// TwinCAT 3 PLC project GattSim
// ProgramVersion: 3.1.4022.3
// libraries:
//   Tc2_Standard, * (Beckhoff Automation GmbH)
//   Tc2_System, * (Beckhoff Automation GmbH)
//   Tc2_Utilities, * (Beckhoff Automation GmbH)
//   Tc3_Module, * (Beckhoff Automation GmbH)
//   Vacuum System Simulator Library, * (SLAC)
// project tree:
//   GVLs/ GVL_GATT.TcGVL, GVL_Variables.TcGVL
//   / PlcTask.TcTTO, SimTask.TcTTO
//   POUs/ MAIN.TcPOU, PRG_DIAGNOSTIC.TcPOU, PRG_GATT.TcPOU
// (motion and I/O tree: see PLC project gattplc)
// real-time tasks:
//   TASK PlcTask: cycle T#10ms, priority 20, ADS port 350
//   TASK SimTask: cycle T#10ms, priority 21, ADS port 351

CONFIGURATION GattSim
    RESOURCE PLC ON TwinCAT3
        TASK PlcTask(INTERVAL := T#10ms, PRIORITY := 20);
        TASK SimTask(INTERVAL := T#10ms, PRIORITY := 21);
        PROGRAM MAIN WITH SimTask : MAIN;
    END_RESOURCE
END_CONFIGURATION

// ---- GVLs/GVL_GATT.TcGVL
VAR_GLOBAL


// ST_Volume

st_AT1K0_GAS_VRC_10_VOL : ST_Volume := (rVolume := 1E3, rPressure := Global_Pressure, rVLeak := Global_Leak);
st_AT1K0_GAS_PTM_10_VOL : ST_Volume := (rVolume := 1E3, rPressure := Global_Pressure, rVLeak := Global_Leak);
st_GATT : ST_Volume := (rVolume := 1E3, rPressure := Global_Pressure, rVLeak := Global_Leak);
st_AT1K0_GAS_VRC_20_VOL : ST_Volume := (rVolume := 1E3, rPressure := Global_Pressure, rVLeak := Global_Leak);
st_AT1K0_GAS_VRC_30_VOL : ST_Volume := (rVolume := 1E3, rPressure := Global_Pressure, rVLeak := Global_Leak);
st_AT1K0_GAS_VRC_40_VOL : ST_Volume := (rVolume := 1E3, rPressure := Global_Pressure, rVLeak := Global_Leak);
st_AT1K0_GAS_VRC_50_VOL : ST_Volume := (rVolume := 1E3, rPressure := Global_Pressure, rVLeak := Global_Leak);
st_AT1K0_GAS_VGP_80_VOL : ST_Volume := (rVolume := 1E3, rPressure := Global_Pressure, rVLeak := Global_Leak);
st_BypassLine2 : ST_Volume := (rVolume := 1E3, rPressure := Global_Pressure, rVLeak := Global_Leak);
st_BypassLine1 : ST_Volume := (rVolume := 1E3, rPressure := Global_Pressure, rVLeak := Global_Leak);
st_AT1K0_GAS_VRC_100_VOL : ST_Volume := (rVolume := 1E3, rPressure := Global_Pressure, rVLeak := Global_Leak);
st_AT1K0_GAS_VRC_110_VOL : ST_Volume := (rVolume := 1E3, rPressure := Global_Pressure, rVLeak := Global_Leak);
st_AT1K0_GAS_PTM_120_VOL : ST_Volume := (rVolume := 1E3, rPressure := Global_Pressure, rVLeak := Global_Leak);
st_AT1K0_GAS_VRC_120_VOL : ST_Volume := (rVolume := 1E3, rPressure := Global_Pressure, rVLeak := Global_Leak);
st_AT1K0_GAS_VRC_130_VOL : ST_Volume := (rVolume := 1E3, rPressure := Global_Pressure, rVLeak := Global_Leak);
st_AT1K0_GAS_PTM_140_VOL : ST_Volume := (rVolume := 1E3, rPressure := Global_Pressure, rVLeak := Global_Leak);
st_AT1K0_GAS_VRC_140_VOL : ST_Volume := (rVolume := 1E3, rPressure := Global_Pressure, rVLeak := Global_Leak);

// ST_MechPump

st_AT1K0_GAS_PTM_10 : ST_MechPump := (iMaxSpd:=1000, rBasePress:=1E-9, rMaxLoad:=0.95);
st_AT1K0_GAS_PTM_20 : ST_MechPump := (iMaxSpd:=1000, rBasePress:=1E-9, rMaxLoad:=0.95);
st_AT1K0_GAS_PMF_10 : ST_MechPump := (rMRE:=10, rBasePress:=1E-3);
st_AT1K0_GAS_PTM_30 : ST_MechPump := (iMaxSpd:=1000, rBasePress:=1E-9, rMaxLoad:=0.95);
st_AT1K0_GAS_PTM_40 : ST_MechPump := (iMaxSpd:=1000, rBasePress:=1E-9, rMaxLoad:=0.95);
st_AT1K0_GAS_PMF_60 : ST_MechPump := (rMRE:=10, rBasePress:=1E-3);
st_AT1K0_GAS_PTM_80 : ST_MechPump := (iMaxSpd:=1000, rBasePress:=1E-9, rMaxLoad:=0.95);
st_AT1K0_GAS_PTM_110 : ST_MechPump := (iMaxSpd:=1000, rBasePress:=1E-9, rMaxLoad:=0.95);
st_AT1K0_GAS_PTM_120 : ST_MechPump := (iMaxSpd:=1000, rBasePress:=1E-9, rMaxLoad:=0.95);
st_AT1K0_GAS_PTM_130 : ST_MechPump := (iMaxSpd:=1000, rBasePress:=1E-9, rMaxLoad:=0.95);
st_AT1K0_GAS_PTM_140 : ST_MechPump := (iMaxSpd:=1000, rBasePress:=1E-9, rMaxLoad:=0.95);

// FB_TurboPump

fb_AT1K0_GAS_PTM_10 : FB_TurboPump;
fb_AT1K0_GAS_PTM_20 : FB_TurboPump;
fb_AT1K0_GAS_PTM_30 : FB_TurboPump;
fb_AT1K0_GAS_PTM_40 : FB_TurboPump;
fb_AT1K0_GAS_PTM_80 : FB_TurboPump;
fb_AT1K0_GAS_PTM_110 : FB_TurboPump;
fb_AT1K0_GAS_PTM_120 : FB_TurboPump;
fb_AT1K0_GAS_PTM_130 : FB_TurboPump;
fb_AT1K0_GAS_PTM_140 : FB_TurboPump;

// ST_VacuumValve

st_AT1K0_GAS_VRC_10 : ST_VacuumValve := (q_xClsLS := TRUE, q_xOpnLS := FALSE);
st_AT1K0_GAS_VRC_20 : ST_VacuumValve := (q_xClsLS := TRUE, q_xOpnLS := FALSE);
st_AT1K0_GAS_VRC_30 : ST_VacuumValve := (q_xClsLS := TRUE, q_xOpnLS := FALSE);
st_AT1K0_GAS_VRC_40 : ST_VacuumValve := (q_xClsLS := TRUE, q_xOpnLS := FALSE);
st_AT1K0_GAS_VRC_50 : ST_VacuumValve := (q_xClsLS := TRUE, q_xOpnLS := FALSE);
st_AT1K0_GAS_VRC_60 : ST_VacuumValve := (q_xClsLS := TRUE, q_xOpnLS := FALSE);
st_AT1K0_GAS_VRC_90 : ST_VacuumValve := (q_xClsLS := TRUE, q_xOpnLS := FALSE);
st_AT1K0_GAS_VRC_100 : ST_VacuumValve := (q_xClsLS := TRUE, q_xOpnLS := FALSE);
st_AT1K0_GAS_VRC_110 : ST_VacuumValve := (q_xClsLS := TRUE, q_xOpnLS := FALSE);
st_AT1K0_GAS_VRC_120 : ST_VacuumValve := (q_xClsLS := TRUE, q_xOpnLS := FALSE);
st_AT1K0_GAS_VRC_130 : ST_VacuumValve := (q_xClsLS := TRUE, q_xOpnLS := FALSE);
st_AT1K0_GAS_VRC_140 : ST_VacuumValve := (q_xClsLS := TRUE, q_xOpnLS := FALSE);

// FB_VacuumValve

fb_AT1K0_GAS_VRC_10 : FB_VacuumValve;
fb_AT1K0_GAS_VRC_20 : FB_VacuumValve;
fb_AT1K0_GAS_VRC_30 : FB_VacuumValve;
fb_AT1K0_GAS_VRC_40 : FB_VacuumValve;
fb_AT1K0_GAS_VRC_50 : FB_VacuumValve;
fb_AT1K0_GAS_VRC_60 : FB_VacuumValve;
fb_AT1K0_GAS_VRC_90 : FB_VacuumValve;
fb_AT1K0_GAS_VRC_100 : FB_VacuumValve;
fb_AT1K0_GAS_VRC_110 : FB_VacuumValve;
fb_AT1K0_GAS_VRC_120 : FB_VacuumValve;
fb_AT1K0_GAS_VRC_130 : FB_VacuumValve;
fb_AT1K0_GAS_VRC_140 : FB_VacuumValve;

// ST_MKS_275

st_AT1K0_GAS_GPI_10 : ST_MKS_275 := (q_xGaugeConnected := TRUE);
st_AT1K0_GAS_GPI_20 : ST_MKS_275 := (q_xGaugeConnected := TRUE);
st_AT1K0_GAS_GPI_11 : ST_MKS_275 := (q_xGaugeConnected := TRUE);
st_AT1K0_GAS_GPI_30 : ST_MKS_275 := (q_xGaugeConnected := TRUE);
st_AT1K0_GAS_GPI_40 : ST_MKS_275 := (q_xGaugeConnected := TRUE);
st_AT1K0_GAS_GPI_50 : ST_MKS_275 := (q_xGaugeConnected := TRUE);
st_AT1K0_GAS_GPI_60 : ST_MKS_275 := (q_xGaugeConnected := TRUE);
st_AT1K0_GAS_GPI_51 : ST_MKS_275 := (q_xGaugeConnected := TRUE);
st_AT1K0_GAS_GPI_80 : ST_MKS_275 := (q_xGaugeConnected := TRUE);
st_AT1K0_GAS_GPI_90 : ST_MKS_275 := (q_xGaugeConnected := TRUE);
st_AT1K0_GAS_GPI_100 : ST_MKS_275 := (q_xGaugeConnected := TRUE);
st_FEES_GATT_GPI_111 : ST_MKS_275 := (q_xGaugeConnected := TRUE);
st_AT1K0_GAS_GPI_110 : ST_MKS_275 := (q_xGaugeConnected := TRUE);
st_AT1K0_GAS_GPI_121 : ST_MKS_275 := (q_xGaugeConnected := TRUE);
st_AT1K0_GAS_GPI_120 : ST_MKS_275 := (q_xGaugeConnected := TRUE);
st_AT1K0_GAS_GPI_130 : ST_MKS_275 := (q_xGaugeConnected := TRUE);
st_AT1K0_GAS_GPI_141 : ST_MKS_275 := (q_xGaugeConnected := TRUE);
st_AT1K0_GAS_GPI_140 : ST_MKS_275 := (q_xGaugeConnected := TRUE);

// FB_MKS_275

fb_AT1K0_GAS_GPI_10 : FB_MKS_275;
fb_AT1K0_GAS_GPI_20 : FB_MKS_275;
fb_AT1K0_GAS_GPI_11 : FB_MKS_275;
fb_AT1K0_GAS_GPI_30 : FB_MKS_275;
fb_AT1K0_GAS_GPI_40 : FB_MKS_275;
fb_AT1K0_GAS_GPI_50 : FB_MKS_275;
fb_AT1K0_GAS_GPI_60 : FB_MKS_275;
fb_AT1K0_GAS_GPI_51 : FB_MKS_275;
fb_AT1K0_GAS_GPI_80 : FB_MKS_275;
fb_AT1K0_GAS_GPI_90 : FB_MKS_275;
fb_AT1K0_GAS_GPI_100 : FB_MKS_275;
fb_FEES_GATT_GPI_111 : FB_MKS_275;
fb_AT1K0_GAS_GPI_110 : FB_MKS_275;
fb_AT1K0_GAS_GPI_121 : FB_MKS_275;
fb_AT1K0_GAS_GPI_120 : FB_MKS_275;
fb_AT1K0_GAS_GPI_130 : FB_MKS_275;
fb_AT1K0_GAS_GPI_141 : FB_MKS_275;
fb_AT1K0_GAS_GPI_140 : FB_MKS_275;

// ST_MKS_422

st_AT1K0_GAS_GCC_10 : ST_MKS_422 := (q_xGaugeConnected := TRUE);
st_AT1K0_GAS_GCC_20 : ST_MKS_422 := (q_xGaugeConnected := TRUE);
st_AT1K0_GAS_GCC_30 : ST_MKS_422 := (q_xGaugeConnected := TRUE);
st_AT1K0_GAS_GCC_40 : ST_MKS_422 := (q_xGaugeConnected := TRUE);
st_AT1K0_GAS_GCC_50 : ST_MKS_422 := (q_xGaugeConnected := TRUE);
st_AT1K0_GAS_GCC_60 : ST_MKS_422 := (q_xGaugeConnected := TRUE);
st_AT1K0_GAS_GCC_80 : ST_MKS_422 := (q_xGaugeConnected := TRUE);
st_AT1K0_GAS_GCC_90 : ST_MKS_422 := (q_xGaugeConnected := TRUE);
st_AT1K0_GAS_GCC_100 : ST_MKS_422 := (q_xGaugeConnected := TRUE);
st_AT1K0_GAS_GCC_110 : ST_MKS_422 := (q_xGaugeConnected := TRUE);
st_AT1K0_GAS_GCC_120 : ST_MKS_422 := (q_xGaugeConnected := TRUE);
st_AT1K0_GAS_GCC_130 : ST_MKS_422 := (q_xGaugeConnected := TRUE);
st_AT1K0_GAS_GCC_140 : ST_MKS_422 := (q_xGaugeConnected := TRUE);

// FB_MKS_422

fb_AT1K0_GAS_GCC_10 : FB_MKS_422;
fb_AT1K0_GAS_GCC_20 : FB_MKS_422;
fb_AT1K0_GAS_GCC_30 : FB_MKS_422;
fb_AT1K0_GAS_GCC_40 : FB_MKS_422;
fb_AT1K0_GAS_GCC_50 : FB_MKS_422;
fb_AT1K0_GAS_GCC_60 : FB_MKS_422;
fb_AT1K0_GAS_GCC_80 : FB_MKS_422;
fb_AT1K0_GAS_GCC_90 : FB_MKS_422;
fb_AT1K0_GAS_GCC_100 : FB_MKS_422;
fb_AT1K0_GAS_GCC_110 : FB_MKS_422;
fb_AT1K0_GAS_GCC_120 : FB_MKS_422;
fb_AT1K0_GAS_GCC_130 : FB_MKS_422;
fb_AT1K0_GAS_GCC_140 : FB_MKS_422;

// FB_RoughPump

fb_AT1K0_GAS_PMF_10 : FB_RoughPump;
fb_AT1K0_GAS_PMF_60 : FB_RoughPump;

END_VAR

// ---- GVLs/GVL_Variables.TcGVL
{attribute 'global_init_slot' := '40500'} // make sure variables are initialized before other GVLs
VAR_GLOBAL

Global_Leak : REAL := 0;
Global_Pressure : REAL := 0.0079;
New_Pressure : REAL := 22.0; //Torr
Global_OverridePressure : BOOL := FALSE;

END_VAR

// ---- POUs/MAIN.TcPOU
PROGRAM MAIN
VAR
END_VAR

PRG_DIAGNOSTIC();
PRG_GATT();

END_PROGRAM

// ---- POUs/PRG_DIAGNOSTIC.TcPOU
PROGRAM PRG_DIAGNOSTIC
VAR
   heartbeat AT %Q* : UINT := 0;
END_VAR

heartbeat := heartbeat + 1;
IF heartbeat > 65000
   THEN heartbeat := 0;
END_IF

END_PROGRAM

// ---- POUs/PRG_GATT.TcPOU
PROGRAM PRG_GATT
VAR
END_VAR


// FB_TurboPump

fb_AT1K0_GAS_PTM_10(stVlInlet := st_AT1K0_GAS_VRC_10_VOL, stVlOutlet := st_AT1K0_GAS_PTM_10_VOL, stPump := st_AT1K0_GAS_PTM_10);
fb_AT1K0_GAS_PTM_20(stVlInlet := st_AT1K0_GAS_VRC_20_VOL, stVlOutlet := st_AT1K0_GAS_PTM_10_VOL, stPump := st_AT1K0_GAS_PTM_20);
fb_AT1K0_GAS_PTM_30(stVlInlet := st_AT1K0_GAS_VRC_30_VOL, stVlOutlet := st_AT1K0_GAS_PTM_10_VOL, stPump := st_AT1K0_GAS_PTM_30);
fb_AT1K0_GAS_PTM_40(stVlInlet := st_AT1K0_GAS_VRC_40_VOL, stVlOutlet := st_AT1K0_GAS_PTM_10_VOL, stPump := st_AT1K0_GAS_PTM_40);
fb_AT1K0_GAS_PTM_80(stVlInlet := st_AT1K0_GAS_VGP_80_VOL, stVlOutlet := st_BypassLine2, stPump := st_AT1K0_GAS_PTM_80);
fb_AT1K0_GAS_PTM_110(stVlInlet := st_AT1K0_GAS_VRC_110_VOL, stVlOutlet := st_BypassLine2, stPump := st_AT1K0_GAS_PTM_110);
fb_AT1K0_GAS_PTM_120(stVlInlet := st_AT1K0_GAS_VRC_120_VOL, stVlOutlet := st_AT1K0_GAS_PTM_120_VOL, stPump := st_AT1K0_GAS_PTM_120);
fb_AT1K0_GAS_PTM_130(stVlInlet := st_AT1K0_GAS_VRC_130_VOL, stVlOutlet := st_AT1K0_GAS_PTM_120_VOL, stPump := st_AT1K0_GAS_PTM_130);
fb_AT1K0_GAS_PTM_140(stVlInlet := st_AT1K0_GAS_VRC_140_VOL, stVlOutlet := st_AT1K0_GAS_PTM_140_VOL, stPump := st_AT1K0_GAS_PTM_140);

// FB_VacuumValve

fb_AT1K0_GAS_VRC_10(stAVol := st_GATT, stBvol := st_AT1K0_GAS_VRC_10_VOL, stValve := st_AT1K0_GAS_VRC_10);
fb_AT1K0_GAS_VRC_20(stAVol := st_GATT, stBvol := st_AT1K0_GAS_VRC_20_VOL, stValve := st_AT1K0_GAS_VRC_20);
fb_AT1K0_GAS_VRC_30(stAVol := st_GATT, stBvol := st_AT1K0_GAS_VRC_30_VOL, stValve := st_AT1K0_GAS_VRC_30);
fb_AT1K0_GAS_VRC_40(stAVol := st_GATT, stBvol := st_AT1K0_GAS_VRC_40_VOL, stValve := st_AT1K0_GAS_VRC_40);
fb_AT1K0_GAS_VRC_50(stAVol := st_GATT, stBvol := st_AT1K0_GAS_VRC_50_VOL, stValve := st_AT1K0_GAS_VRC_50);
fb_AT1K0_GAS_VRC_60(stAVol := st_GATT, stBvol := st_AT1K0_GAS_VRC_50_VOL, stValve := st_AT1K0_GAS_VRC_60);
fb_AT1K0_GAS_VRC_90(stAVol := st_GATT, stBvol := st_BypassLine1, stValve := st_AT1K0_GAS_VRC_90);
fb_AT1K0_GAS_VRC_100(stAVol := st_GATT, stBvol := st_AT1K0_GAS_VRC_100_VOL, stValve := st_AT1K0_GAS_VRC_100);
fb_AT1K0_GAS_VRC_110(stAVol := st_GATT, stBvol := st_AT1K0_GAS_VRC_110_VOL, stValve := st_AT1K0_GAS_VRC_110);
fb_AT1K0_GAS_VRC_120(stAVol := st_GATT, stBvol := st_AT1K0_GAS_VRC_120_VOL, stValve := st_AT1K0_GAS_VRC_120);
fb_AT1K0_GAS_VRC_130(stAVol := st_GATT, stBvol := st_AT1K0_GAS_VRC_130_VOL, stValve := st_AT1K0_GAS_VRC_130);
fb_AT1K0_GAS_VRC_140(stAVol := st_GATT, stBvol := st_AT1K0_GAS_VRC_140_VOL, stValve := st_AT1K0_GAS_VRC_140);

// FB_MKS_275

fb_AT1K0_GAS_GPI_10(stVolume := st_GATT, stGauge := st_AT1K0_GAS_GPI_10);
fb_AT1K0_GAS_GPI_20(stVolume := st_GATT, stGauge := st_AT1K0_GAS_GPI_20);
fb_AT1K0_GAS_GPI_11(stVolume := st_AT1K0_GAS_PTM_10_VOL, stGauge := st_AT1K0_GAS_GPI_11);
fb_AT1K0_GAS_GPI_30(stVolume := st_GATT, stGauge := st_AT1K0_GAS_GPI_30);
fb_AT1K0_GAS_GPI_40(stVolume := st_GATT, stGauge := st_AT1K0_GAS_GPI_40);
fb_AT1K0_GAS_GPI_50(stVolume := st_GATT, stGauge := st_AT1K0_GAS_GPI_50);
fb_AT1K0_GAS_GPI_60(stVolume := st_GATT, stGauge := st_AT1K0_GAS_GPI_60);
fb_AT1K0_GAS_GPI_51(stVolume := st_AT1K0_GAS_VRC_50_VOL, stGauge := st_AT1K0_GAS_GPI_51);
fb_AT1K0_GAS_GPI_80(stVolume := st_GATT, stGauge := st_AT1K0_GAS_GPI_80);
fb_AT1K0_GAS_GPI_90(stVolume := st_GATT, stGauge := st_AT1K0_GAS_GPI_90);
fb_AT1K0_GAS_GPI_100(stVolume := st_GATT, stGauge := st_AT1K0_GAS_GPI_100);
fb_FEES_GATT_GPI_111(stVolume := st_BypassLine2, stGauge := st_FEES_GATT_GPI_111);
fb_AT1K0_GAS_GPI_110(stVolume := st_GATT, stGauge := st_AT1K0_GAS_GPI_110);
fb_AT1K0_GAS_GPI_121(stVolume := st_AT1K0_GAS_PTM_120_VOL, stGauge := st_AT1K0_GAS_GPI_121);
fb_AT1K0_GAS_GPI_120(stVolume := st_GATT, stGauge := st_AT1K0_GAS_GPI_120);
fb_AT1K0_GAS_GPI_130(stVolume := st_GATT, stGauge := st_AT1K0_GAS_GPI_130);
fb_AT1K0_GAS_GPI_141(stVolume := st_AT1K0_GAS_PTM_140_VOL, stGauge := st_AT1K0_GAS_GPI_141);
fb_AT1K0_GAS_GPI_140(stVolume := st_GATT, stGauge := st_AT1K0_GAS_GPI_140);

// FB_MKS_422

fb_AT1K0_GAS_GCC_10(stVolume := st_GATT, stGauge := st_AT1K0_GAS_GCC_10);
fb_AT1K0_GAS_GCC_20(stVolume := st_GATT, stGauge := st_AT1K0_GAS_GCC_20);
fb_AT1K0_GAS_GCC_30(stVolume := st_GATT, stGauge := st_AT1K0_GAS_GCC_30);
fb_AT1K0_GAS_GCC_40(stVolume := st_GATT, stGauge := st_AT1K0_GAS_GCC_40);
fb_AT1K0_GAS_GCC_50(stVolume := st_GATT, stGauge := st_AT1K0_GAS_GCC_50);
fb_AT1K0_GAS_GCC_60(stVolume := st_GATT, stGauge := st_AT1K0_GAS_GCC_60);
fb_AT1K0_GAS_GCC_80(stVolume := st_GATT, stGauge := st_AT1K0_GAS_GCC_80);
fb_AT1K0_GAS_GCC_90(stVolume := st_GATT, stGauge := st_AT1K0_GAS_GCC_90);
fb_AT1K0_GAS_GCC_100(stVolume := st_GATT, stGauge := st_AT1K0_GAS_GCC_100);
fb_AT1K0_GAS_GCC_110(stVolume := st_GATT, stGauge := st_AT1K0_GAS_GCC_110);
fb_AT1K0_GAS_GCC_120(stVolume := st_GATT, stGauge := st_AT1K0_GAS_GCC_120);
fb_AT1K0_GAS_GCC_130(stVolume := st_GATT, stGauge := st_AT1K0_GAS_GCC_130);
fb_AT1K0_GAS_GCC_140(stVolume := st_GATT, stGauge := st_AT1K0_GAS_GCC_140);

// FB_RoughPump

fb_AT1K0_GAS_PMF_10(stVolInlet := st_AT1K0_GAS_PTM_10_VOL, stPump := st_AT1K0_GAS_PMF_10);
fb_AT1K0_GAS_PMF_60(stVolInlet := st_AT1K0_GAS_VRC_50_VOL, stPump := st_AT1K0_GAS_PMF_60);

END_PROGRAM
